KUKA KRL program: wkz2_stb_ab.src, wkz2_stb_ab.dat

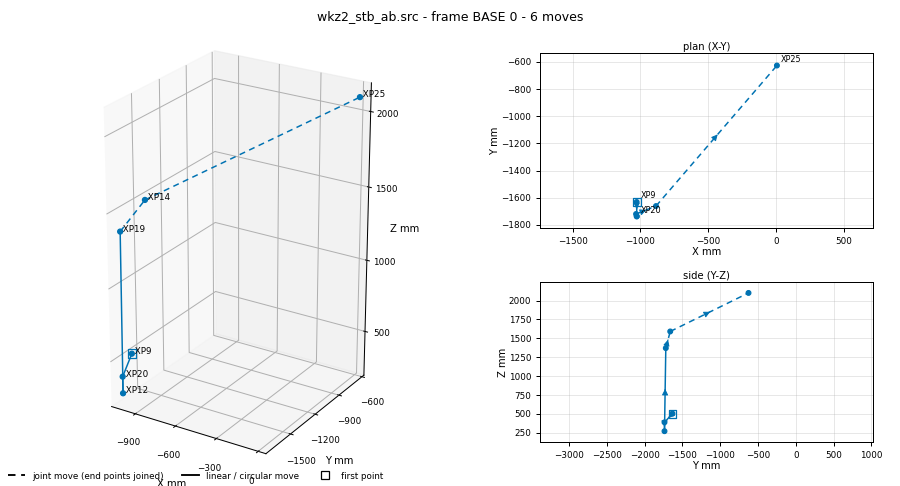
[picture p0: tool path of wkz2_stb_ab.src in frame BASE 0, 6 of 6 moves have a stored position in this frame; points joined in program order, loops and branches not executed]
--- wkz2_stb_ab.src ---
&ACCESS RVO
&REL 1
&COMMENT Deposito GUN C1_STB
&PARAM DISKPATH = KRC:\R1\Program
&PARAM TEMPLATE = C:\KRC\Roboter\Template\vorgabe
&PARAM EDITMASK = *
DEF wkz2_stb_ab( )
;FOLD INI
  ;FOLD BASISTECH INI
    GLOBAL INTERRUPT DECL 3 WHEN $STOPMESS==TRUE DO IR_STOPM ( )
    INTERRUPT ON 3
    BAS (#INITMOV,0 )
  ;ENDFOLD (BASISTECH INI)
;FOLD GRIPPERTECH INI
USER_GRP(0,DUMMY,DUMMY,GDEFAULT)
;ENDFOLD (GRIPPERTECH INI)
  ;FOLD USER INI
    ;Make your modifications here

  ;ENDFOLD (USER INI)
;ENDFOLD (INI)

; Caracterização dos meios de produção:
; Versão Atual:
; 08/06/2013 12:00 Name: P13.050-R1 CHANGES: Deposita gun C1
; (F2 6640 0018 984)

chk_w2_wechs_ok() ; check c1

$advance=3

;FOLD WAIT FOR ( IN 219 'Posicao p/ Acoplamento OK' );%{PE}%R 8.2.20,%MKUKATPBASIS,%CEXT_WAIT_FOR,%VEXT_WAIT_FOR,%P 2:, 4:, 5:$IN, 6:219, 7:Posicao p/ Acoplamento OK, 9:
WAIT FOR  ( $IN[219] )
;ENDFOLD
;FOLD WAIT FOR NOT ( IN 209 'DOCK 7 Deposito Ocupado' );%{PE}%R 8.2.20,%MKUKATPBASIS,%CEXT_WAIT_FOR,%VEXT_WAIT_FOR,%P 2:NOT, 4:, 5:$IN, 6:209, 7:DOCK 7 Deposito Ocupado, 9:
WAIT FOR  NOT ( $IN[209] )
;ENDFOLD
;FOLD WAIT FOR ( IN 213 'DOCK 7 Proteção Aberta' );%{PE}%R 8.2.20,%MKUKATPBASIS,%CEXT_WAIT_FOR,%VEXT_WAIT_FOR,%P 2:, 4:, 5:$IN, 6:213, 7:DOCK 7 Proteção Aberta, 9:
WAIT FOR  ( $IN[213] )
;ENDFOLD
;FOLD WAIT FOR NOT ( IN 214 'DOCK 7 Proteção Fechada' );%{PE}%R 8.2.20,%MKUKATPBASIS,%CEXT_WAIT_FOR,%VEXT_WAIT_FOR,%P 2:NOT, 4:, 5:$IN, 6:214, 7:DOCK 7 Proteção Fechada, 9:
WAIT FOR  NOT ( $IN[214] )
;ENDFOLD

;FOLD PTP P9 CONT Vel=100 % PDAT7 Tool[2]:GUN C1 Base[2]:Accelo;%{PE}%R 8.2.20,%MKUKATPBASIS,%CMOVE,%VPTP,%P 1:PTP, 2:P9, 3:C_DIS, 5:100, 7:PDAT7
$BWDSTART=FALSE
PDAT_ACT=PPDAT7
FDAT_ACT=FP9
BAS(#PTP_PARAMS,100)
PTP XP9 C_DIS
;ENDFOLD

;FOLD LIN P20 Vel=2 m/s CPDAT14 Tool[2]:GUN C1 Base[0];%{PE}%R 8.2.20,%MKUKATPBASIS,%CMOVE,%VLIN,%P 1:LIN, 2:P20, 3:, 5:2, 7:CPDAT14
$BWDSTART=FALSE
LDAT_ACT=LCPDAT14
FDAT_ACT=FP20
BAS(#CP_PARAMS,2)
LIN XP20
;ENDFOLD

;FOLD ; PONTO DE DEPOSITO DA PINCA;%{PE}%R 8.2.19,%MKUKATPBASIS,%CCOMMENT,%VNORMAL,%P 2:PONTO  DE  DEPOSITO  DA  PINCA
;ENDFOLD
;FOLD LIN P12 Vel=0.5 m/s CPDAT9 Tool[2]:GUN C1 Base[0];%{PE}%R 8.2.20,%MKUKATPBASIS,%CMOVE,%VLIN,%P 1:LIN, 2:P12, 3:, 5:0.5, 7:CPDAT9
$BWDSTART=FALSE
LDAT_ACT=LCPDAT9
FDAT_ACT=FP12
BAS(#CP_PARAMS,0.5)
LIN XP12
;ENDFOLD

;FOLD WAIT FOR ( IN 209 'DOCK 7 Deposito Ocupado' );%{PE}%R 8.2.20,%MKUKATPBASIS,%CEXT_WAIT_FOR,%VEXT_WAIT_FOR,%P 2:, 4:, 5:$IN, 6:209, 7:DOCK 7 Deposito Ocupado, 9:
WAIT FOR  ( $IN[209] )
;ENDFOLD
;FOLD WAIT FOR ( IN 222 'Liberacao p/ Desbloqueio' );%{PE}%R 8.2.20,%MKUKATPBASIS,%CEXT_WAIT_FOR,%VEXT_WAIT_FOR,%P 2:, 4:, 5:$IN, 6:222, 7:Liberacao p/ Desbloqueio, 9:
WAIT FOR  ( $IN[222] )
;ENDFOLD
;FOLD OUT 224 'Bloquear MPS' State=FALSE ;%{PE}%R 8.2.20,%MKUKATPBASIS,%COUT,%VOUTX,%P 2:224, 3:Bloquear MPS, 5:FALSE, 6:
$OUT[224]=FALSE
;ENDFOLD
;FOLD OUT 223 'Desbloquear MPS' State=TRUE ;%{PE}%R 8.2.20,%MKUKATPBASIS,%COUT,%VOUTX,%P 2:223, 3:Desbloquear MPS, 5:TRUE, 6:
$OUT[223]=TRUE
;ENDFOLD
;FOLD WAIT FOR ( IN 217 'MPS Destravado' );%{PE}%R 8.2.20,%MKUKATPBASIS,%CEXT_WAIT_FOR,%VEXT_WAIT_FOR,%P 2:, 4:, 5:$IN, 6:217, 7:MPS Destravado, 9:
WAIT FOR  ( $IN[217] )
;ENDFOLD
;FOLD WAIT FOR NOT ( IN 221 'MPS Travado' );%{PE}%R 8.2.20,%MKUKATPBASIS,%CEXT_WAIT_FOR,%VEXT_WAIT_FOR,%P 2:NOT, 4:, 5:$IN, 6:221, 7:MPS Travado, 9:
WAIT FOR  NOT ( $IN[221] )
;ENDFOLD
;FOLD WAIT Time=0.25 sec;%{PE}%R 8.2.20,%MKUKATPBASIS,%CWAIT,%VWAIT,%P 3:0.25
WAIT SEC 0.25
;ENDFOLD
;FOLD IBUS OFF;%{PE}%R 8.2.20,%MKUKATPBASIS,%CIBUS,%VMAP,%P 2:#OFF, 3:2
$IBUS_OFF=$IBUS_ON
$IBUS_ON=0
;ENDFOLD
;FOLD WAIT Time=0.25 sec;%{PE}%R 8.2.20,%MKUKATPBASIS,%CWAIT,%VWAIT,%P 3:0.25
WAIT SEC 0.25
;ENDFOLD

;FOLD LIN P19 Vel=1 m/s CPDAT13 Tool[8]:TOOL_CHANGER Base[0];%{PE}%R 8.2.20,%MKUKATPBASIS,%CMOVE,%VLIN,%P 1:LIN, 2:P19, 3:, 5:1, 7:CPDAT13
$BWDSTART=FALSE
LDAT_ACT=LCPDAT13
FDAT_ACT=FP19
BAS(#CP_PARAMS,1)
LIN XP19
;ENDFOLD

;FOLD WAIT FOR ( IN 209 'DOCK 7 Deposito Ocupado' ) CONT;%{PE}%R 8.2.20,%MKUKATPBASIS,%CEXT_WAIT_FOR,%VEXT_WAIT_FOR,%P 2:, 4:, 5:$IN, 6:209, 7:DOCK 7 Deposito Ocupado, 9:CONTINUE
CONTINUE
WAIT FOR  ( $IN[209] )
;ENDFOLD
;FOLD WAIT FOR NOT ( IN 219 'Posicao p/ Acoplamento OK' ) CONT;%{PE}%R 8.2.20,%MKUKATPBASIS,%CEXT_WAIT_FOR,%VEXT_WAIT_FOR,%P 2:NOT, 4:, 5:$IN, 6:219, 7:Posicao p/ Acoplamento OK, 9:CONTINUE
CONTINUE
WAIT FOR  NOT ( $IN[219] )
;ENDFOLD
;FOLD OUT 223 'Desbloquear MPS' State=FALSE CONT;%{PE}%R 8.2.20,%MKUKATPBASIS,%COUT,%VOUTX,%P 2:223, 3:Desbloquear MPS, 5:FALSE, 6:CONTINUE
CONTINUE
$OUT[223]=FALSE
;ENDFOLD

;FOLD PTP P14 CONT Vel=100 % PDAT8 Tool[2]:GUN C1 Base[2]:Accelo;%{PE}%R 8.2.20,%MKUKATPBASIS,%CMOVE,%VPTP,%P 1:PTP, 2:P14, 3:C_DIS, 5:100, 7:PDAT8
$BWDSTART=FALSE
PDAT_ACT=PPDAT8
FDAT_ACT=FP14
BAS(#PTP_PARAMS,100)
PTP XP14 C_DIS
;ENDFOLD
;FOLD PTP P25 Vel=100 % PDAT13 Tool[8]:TOOL_CHANGER Base[0];%{PE}%R 8.2.20,%MKUKATPBASIS,%CMOVE,%VPTP,%P 1:PTP, 2:P25, 3:, 5:100, 7:PDAT13
$BWDSTART=FALSE
PDAT_ACT=PPDAT13
FDAT_ACT=FP25
BAS(#PTP_PARAMS,100)
PTP XP25
;ENDFOLD

;FOLD PULSE 216 'DOCK 7 Fechar Proteção' State=TRUE Time=0.5 sec;%{PE}%R 8.2.20,%MKUKATPBASIS,%COUT,%VPULSE,%P 2:216, 3:DOCK 7 Fechar Proteção, 5:TRUE, 6:, 8:0.5
PULSE($OUT[216], TRUE,0.5)
;ENDFOLD
END

--- wkz2_stb_ab.dat ---
&ACCESS RVO
&REL 1
&COMMENT Deposito GUN C1_STB
&PARAM DISKPATH = KRC:\R1\Program
&PARAM TEMPLATE = C:\KRC\Roboter\Template\vorgabe
&PARAM EDITMASK = *
DEFDAT wkz2_stb_ab
;FOLD EXTERNAL DECLARATIONS;%{PE}%MKUKATPBASIS,%CEXT,%VCOMMON,%P
;FOLD GRIPPERTECH EXT
EXT  H50 (INT  :IN,INT  :IN,INT  :IN,GRP_TYP  :IN )
;ENDFOLD (GRIPPERTECH EXT)
;FOLD SPOTTECH EXT
EXT  USERSPOT (S_COMMAND  :IN,SPOT_TYPE  :IN )
;ENDFOLD (SPOTTECH EXT)
;FOLD BASISTECH EXT;%{PE}%MKUKATPBASIS,%CEXT,%VEXT,%P
EXT  BAS (BAS_COMMAND  :IN,REAL  :IN )
DECL INT SUCCESS
;ENDFOLD (BASISTECH EXT)
;FOLD USER EXT;%{E}%MKUKATPUSER,%CEXT,%VEXT,%P
;Make your modifications here

;ENDFOLD (USER EXT)
;ENDFOLD (EXTERNAL DECLARATIONS)
DECL BASIS_SUGG_T LAST_BASIS={POINT1[] "P0                      ",POINT2[] "P0                      ",CP_PARAMS[] "CPDAT0                  ",PTP_PARAMS[] "PDAT0                   ",CONT[] "                        ",CP_VEL[] "2                       ",PTP_VEL[] " 100                    ",SYNC_PARAMS[] "SYNCDAT                 ",SPL_NAME[] "S0                      "}
DECL E6POS XP9={X -1027.59705,Y -1631.88306,Z 503.879486,A -89.4597702,B -0.808308721,C 0.275945991,S 2,T 10,E1 213.807999,E2 0.0,E3 0.0,E4 0.0,E5 0.0,E6 0.0}
DECL FDAT FP9={TOOL_NO 2,BASE_NO 0,IPO_FRAME #BASE,POINT2[] " ",TQ_STATE FALSE}
DECL E6POS XP12={X -1027.12097,Y -1737.57202,Z 271.306,A -89.4590912,B -0.602925599,C 0.276565105,S 2,T 10,E1 213.207901,E2 0.0,E3 0.0,E4 0.0,E5 0.0,E6 0.0}
DECL FDAT FP12={TOOL_NO 2,BASE_NO 0,IPO_FRAME #BASE,POINT2[] " ",TQ_STATE FALSE}
DECL LDAT LCPDAT9={VEL 2.0,ACC 100.0,APO_DIST 100.0,APO_FAC 50.0,AXIS_VEL 100.0,AXIS_ACC 100.0,ORI_TYP #VAR,CIRC_TYP #BASE,JERK_FAC 50.0,GEAR_JERK 50.0,EXAX_IGN 0}
DECL E6POS XP14={X -885.227417,Y -1661.69202,Z 1591.03296,A -102.484901,B -5.67610502,C 179.018204,S 2,T 10,E1 214.095093,E2 0.0,E3 0.0,E4 0.0,E5 0.0,E6 0.0}
DECL FDAT FP14={TOOL_NO 8,BASE_NO 0,IPO_FRAME #BASE,POINT2[] " ",TQ_STATE FALSE}
DECL E6POS XP19={X -1032.06494,Y -1720.24194,Z 1370.68701,A -74.4582672,B -0.653960884,C -179.888901,S 2,T 10,E1 213.694504,E2 0.0,E3 0.0,E4 0.0,E5 0.0,E6 0.0}
DECL FDAT FP19={TOOL_NO 8,BASE_NO 0,IPO_FRAME #BASE,POINT2[] " ",TQ_STATE FALSE}
DECL LDAT LCPDAT13={VEL 2.0,ACC 100.0,APO_DIST 100.0,APO_FAC 50.0,AXIS_VEL 100.0,AXIS_ACC 100.0,ORI_TYP #VAR,CIRC_TYP #BASE,JERK_FAC 50.0,GEAR_JERK 50.0,EXAX_IGN 0}
DECL E6POS XP20={X -1027.15698,Y -1737.58801,Z 388.610199,A -89.4584274,B -0.603913009,C 0.275392592,S 2,T 10,E1 214.107407,E2 0.0,E3 0.0,E4 0.0,E5 0.0,E6 0.0}
DECL FDAT FP20={TOOL_NO 2,BASE_NO 0,IPO_FRAME #BASE,POINT2[] " ",TQ_STATE FALSE}
DECL LDAT LCPDAT14={VEL 2.0,ACC 100.0,APO_DIST 50.0,APO_FAC 50.0,AXIS_VEL 100.0,AXIS_ACC 100.0,ORI_TYP #VAR,CIRC_TYP #BASE,JERK_FAC 50.0,GEAR_JERK 50.0,EXAX_IGN 0}
DECL PDAT PPDAT7={VEL 100.0,ACC 100.0,APO_DIST 50.0,APO_MODE #CDIS}
DECL PDAT PPDAT8={VEL 100.0,ACC 100.0,APO_DIST 50.0,APO_MODE #CDIS}
DECL E6POS XP25={X 5.94878006,Y -626.062073,Z 2100.46289,A -77.0247192,B -9.68836498,C 176.383804,S 2,T 2,E1 213.667801,E2 0.0,E3 0.0,E4 0.0,E5 0.0,E6 0.0}
DECL FDAT FP25={TOOL_NO 8,BASE_NO 0,IPO_FRAME #BASE,POINT2[] " ",TQ_STATE FALSE}
DECL PDAT PPDAT13={VEL 100.0,ACC 100.0,APO_DIST 100.0,APO_MODE #CDIS}
ENDDAT
